PROGRAM Stn052_20_ReceivingBreakStopsGrn
VAR
	
//(1 omitted intentially, 3LnSw using this location)	
//		.fbBreakStop[1].iBufferFull :=  <0,1,0>TIIB[N21S00 (AL1332)]^N21S03 (AL2341)^TxPDO^input byte 2;
//		.fbBreakStop[1].iPuckPresent :=  <0,1,0>TIIB[N21S00 (AL1332)]^N21S03 (AL2341)^TxPDO^input byte 0;
//		.fbBreakStop[1].oStopLower :=  <0,1,4>TIIB[N21S00 (AL1332)]^N21S02 (EX260)^RxPDO^output byte 0;
//(3 omitted because the output byte overlaps 2 PLC projects, these are linked in Stn053)
//		.fbBreakStop[31].oStopLower :=  <0,1,0>TIIB[N32S00 (AL1332)]^N32S02 (EX260)^RxPDO^output byte 0;
//		.fbBreakStop[32].oStopLower :=  <0,1,1>TIIB[N32S00 (AL1332)]^N32S02 (EX260)^RxPDO^output byte 0;
//		.fbBreakStop[33].oStopLower :=  <0,1,2>TIIB[N32S00 (AL1332)]^N32S02 (EX260)^RxPDO^output byte 0'}	

	{attribute 'TcLinkToOSO' := '.fbBreakStop[2].iBufferFull :=  <0,1,1>TIIB[N21S00 (AL1332)]^N21S03 (AL2341)^TxPDO^input byte 2;
		.fbBreakStop[2].iPuckPresent :=  <0,1,1>TIIB[N21S00 (AL1332)]^N21S03 (AL2341)^TxPDO^input byte 0;
		.fbBreakStop[2].oStopLower :=  <0,1,5>TIIB[N21S00 (AL1332)]^N21S02 (EX260)^RxPDO^output byte 0;
		.fbBreakStop[3].iBufferFull :=  <0,1,0>TIIB[N21S00 (AL1332)]^N21S05 (AL2341)^TxPDO^input byte 2;
		.fbBreakStop[3].iPuckPresent :=  <0,1,0>TIIB[N21S00 (AL1332)]^N21S05 (AL2341)^TxPDO^input byte 0;
		.fbBreakStop[3].oStopLower :=  <0,1,6>TIIB[N21S00 (AL1332)]^N21S02 (EX260)^RxPDO^output byte 0;
		.fbBreakStop[4].iBufferFull :=  <0,1,0>TIIB[N26S00 (AL1332)]^N26S01 (AL2341)^TxPDO^input byte 2;
		.fbBreakStop[4].iPuckPresent :=  <0,1,0>TIIB[N26S00 (AL1332)]^N26S01 (AL2341)^TxPDO^input byte 0;
		.fbBreakStop[4].oStopLower :=  <0,1,0>TIIB[N26S00 (AL1332)]^N26S05 (EX260)^RxPDO^output byte 0;
		.fbBreakStop[5].iBufferFull :=  <0,1,2>TIIB[N26S00 (AL1332)]^N26S01 (AL2341)^TxPDO^input byte 2;
		.fbBreakStop[5].iPuckPresent :=  <0,1,2>TIIB[N26S00 (AL1332)]^N26S01 (AL2341)^TxPDO^input byte 0;
		.fbBreakStop[5].oStopLower :=  <0,1,1>TIIB[N26S00 (AL1332)]^N26S05 (EX260)^RxPDO^output byte 0;
		.fbBreakStop[6].iBufferFull :=  <0,1,3>TIIB[N26S00 (AL1332)]^N26S01 (AL2341)^TxPDO^input byte 2;
		.fbBreakStop[6].iPuckPresent :=  <0,1,3>TIIB[N26S00 (AL1332)]^N26S01 (AL2341)^TxPDO^input byte 0;
		.fbBreakStop[6].oStopLower :=  <0,1,4>TIIB[N26S00 (AL1332)]^N26S05 (EX260)^RxPDO^output byte 0;
		.fbBreakStop[7].iBufferFull :=  <0,1,4>TIIB[N26S00 (AL1332)]^N26S01 (AL2341)^TxPDO^input byte 2;
		.fbBreakStop[7].iPuckPresent :=  <0,1,4>TIIB[N26S00 (AL1332)]^N26S01 (AL2341)^TxPDO^input byte 0;
		.fbBreakStop[7].oStopLower :=  <0,1,5>TIIB[N26S00 (AL1332)]^N26S05 (EX260)^RxPDO^output byte 0;
		.fbBreakStop[8].iBufferFull :=  <0,1,0>TIIB[N26S00 (AL1332)]^N26S03 (AL2341)^TxPDO^input byte 2;
		.fbBreakStop[8].iPuckPresent :=  <0,1,0>TIIB[N26S00 (AL1332)]^N26S03 (AL2341)^TxPDO^input byte 0;
		.fbBreakStop[8].oStopLower :=  <0,1,0>TIIB[N26S00 (AL1332)]^N26S06 (EX260)^RxPDO^output byte 0;
		.fbBreakStop[9].iBufferFull :=  <0,1,2>TIIB[N26S00 (AL1332)]^N26S03 (AL2341)^TxPDO^input byte 2;
		.fbBreakStop[9].iPuckPresent :=  <0,1,2>TIIB[N26S00 (AL1332)]^N26S03 (AL2341)^TxPDO^input byte 0;
		.fbBreakStop[9].oStopLower :=  <0,1,1>TIIB[N26S00 (AL1332)]^N26S06 (EX260)^RxPDO^output byte 0;
		.fbBreakStop[10].iBufferFull :=  <0,1,3>TIIB[N26S00 (AL1332)]^N26S03 (AL2341)^TxPDO^input byte 2;
		.fbBreakStop[10].iPuckPresent :=  <0,1,3>TIIB[N26S00 (AL1332)]^N26S03 (AL2341)^TxPDO^input byte 0;
		.fbBreakStop[10].oStopLower :=  <0,1,4>TIIB[N26S00 (AL1332)]^N26S06 (EX260)^RxPDO^output byte 0;
		.fbBreakStop[11].iBufferFull :=  <0,1,4>TIIB[N26S00 (AL1332)]^N26S03 (AL2341)^TxPDO^input byte 2;
		.fbBreakStop[11].iPuckPresent :=  <0,1,4>TIIB[N26S00 (AL1332)]^N26S03 (AL2341)^TxPDO^input byte 0;
		.fbBreakStop[11].oStopLower :=  <0,1,5>TIIB[N26S00 (AL1332)]^N26S06 (EX260)^RxPDO^output byte 0;
		.fbBreakStop[12].iBufferFull :=  <0,1,0>TIIB[N27S00 (AL1332)]^N27S01 (AL2341)^TxPDO^input byte 2;
		.fbBreakStop[12].iPuckPresent :=  <0,1,0>TIIB[N27S00 (AL1332)]^N27S01 (AL2341)^TxPDO^input byte 0;
		.fbBreakStop[12].oStopLower :=  <0,1,0>TIIB[N27S00 (AL1332)]^N27S05 (EX260)^RxPDO^output byte 0;
		.fbBreakStop[13].iBufferFull :=  <0,1,2>TIIB[N27S00 (AL1332)]^N27S01 (AL2341)^TxPDO^input byte 2;
		.fbBreakStop[13].iPuckPresent :=  <0,1,2>TIIB[N27S00 (AL1332)]^N27S01 (AL2341)^TxPDO^input byte 0;
		.fbBreakStop[13].oStopLower :=  <0,1,1>TIIB[N27S00 (AL1332)]^N27S05 (EX260)^RxPDO^output byte 0;
		.fbBreakStop[14].iBufferFull :=  <0,1,3>TIIB[N27S00 (AL1332)]^N27S01 (AL2341)^TxPDO^input byte 2;
		.fbBreakStop[14].iPuckPresent :=  <0,1,3>TIIB[N27S00 (AL1332)]^N27S01 (AL2341)^TxPDO^input byte 0;
		.fbBreakStop[14].oStopLower :=  <0,1,4>TIIB[N27S00 (AL1332)]^N27S05 (EX260)^RxPDO^output byte 0;
		.fbBreakStop[15].iBufferFull :=  <0,1,4>TIIB[N27S00 (AL1332)]^N27S01 (AL2341)^TxPDO^input byte 2;
		.fbBreakStop[15].iPuckPresent :=  <0,1,4>TIIB[N27S00 (AL1332)]^N27S01 (AL2341)^TxPDO^input byte 0;
		.fbBreakStop[15].oStopLower :=  <0,1,5>TIIB[N27S00 (AL1332)]^N27S05 (EX260)^RxPDO^output byte 0;
		.fbBreakStop[16].iBufferFull :=  <0,1,0>TIIB[N27S00 (AL1332)]^N27S03 (AL2341)^TxPDO^input byte 2;
		.fbBreakStop[16].iPuckPresent :=  <0,1,0>TIIB[N27S00 (AL1332)]^N27S03 (AL2341)^TxPDO^input byte 0;
		.fbBreakStop[16].oStopLower :=  <0,1,0>TIIB[N27S00 (AL1332)]^N27S06 (EX260)^RxPDO^output byte 0;
		.fbBreakStop[17].iBufferFull :=  <0,1,2>TIIB[N27S00 (AL1332)]^N27S03 (AL2341)^TxPDO^input byte 2;
		.fbBreakStop[17].iPuckPresent :=  <0,1,2>TIIB[N27S00 (AL1332)]^N27S03 (AL2341)^TxPDO^input byte 0;
		.fbBreakStop[17].oStopLower :=  <0,1,1>TIIB[N27S00 (AL1332)]^N27S06 (EX260)^RxPDO^output byte 0;
		.fbBreakStop[18].iBufferFull :=  <0,1,3>TIIB[N27S00 (AL1332)]^N27S03 (AL2341)^TxPDO^input byte 2;
		.fbBreakStop[18].iPuckPresent :=  <0,1,3>TIIB[N27S00 (AL1332)]^N27S03 (AL2341)^TxPDO^input byte 0;
		.fbBreakStop[18].oStopLower :=  <0,1,4>TIIB[N27S00 (AL1332)]^N27S06 (EX260)^RxPDO^output byte 0;
		.fbBreakStop[19].iBufferFull :=  <0,1,4>TIIB[N27S00 (AL1332)]^N27S03 (AL2341)^TxPDO^input byte 0;
		.fbBreakStop[19].iPuckPresent :=  <0,1,4>TIIB[N27S00 (AL1332)]^N27S03 (AL2341)^TxPDO^input byte 2;
		.fbBreakStop[19].oStopLower :=  <0,1,5>TIIB[N27S00 (AL1332)]^N27S06 (EX260)^RxPDO^output byte 0;
		.fbBreakStop[20].iBufferFull :=  <0,1,3>TIIB[N28S00 (AL1332)]^N28S01 (AL2341)^TxPDO^input byte 2;
		.fbBreakStop[20].iPuckPresent :=  <0,1,3>TIIB[N28S00 (AL1332)]^N28S01 (AL2341)^TxPDO^input byte 0;
		.fbBreakStop[20].oStopLower :=  <0,1,4>TIIB[N28S00 (AL1332)]^N28S05 (EX260)^RxPDO^output byte 0;
		.fbBreakStop[21].iBufferFull :=  <0,1,4>TIIB[N28S00 (AL1332)]^N28S01 (AL2341)^TxPDO^input byte 2;
		.fbBreakStop[21].iPuckPresent :=  <0,1,4>TIIB[N28S00 (AL1332)]^N28S01 (AL2341)^TxPDO^input byte 0;
		.fbBreakStop[21].oStopLower :=  <0,1,5>TIIB[N28S00 (AL1332)]^N28S05 (EX260)^RxPDO^output byte 0;
		.fbBreakStop[22].iBufferFull :=  <0,1,3>TIIB[N28S00 (AL1332)]^N28S03 (AL2341)^TxPDO^input byte 2;
		.fbBreakStop[22].iPuckPresent :=  <0,1,3>TIIB[N28S00 (AL1332)]^N28S03 (AL2341)^TxPDO^input byte 0;
		.fbBreakStop[22].oStopLower :=  <0,1,4>TIIB[N28S00 (AL1332)]^N28S06 (EX260)^RxPDO^output byte 0;
		.fbBreakStop[23].iBufferFull :=  <0,1,4>TIIB[N28S00 (AL1332)]^N28S03 (AL2341)^TxPDO^input byte 2;
		.fbBreakStop[23].iPuckPresent :=  <0,1,4>TIIB[N28S00 (AL1332)]^N28S03 (AL2341)^TxPDO^input byte 0;
		.fbBreakStop[23].oStopLower :=  <0,1,5>TIIB[N28S00 (AL1332)]^N28S06 (EX260)^RxPDO^output byte 0;
		.fbBreakStop[24].iBufferFull :=  <0,1,0>TIIB[N31S00 (AL1332)]^N31S01 (AL2341)^TxPDO^input byte 2;
		.fbBreakStop[24].iPuckPresent :=  <0,1,0>TIIB[N31S00 (AL1332)]^N31S01 (AL2341)^TxPDO^input byte 0;
		.fbBreakStop[24].oStopLower :=  <0,1,0>TIIB[N31S00 (AL1332)]^N31S02 (EX260)^RxPDO^output byte 0;
		.fbBreakStop[25].iBufferFull :=  <0,1,1>TIIB[N31S00 (AL1332)]^N31S01 (AL2341)^TxPDO^input byte 2;
		.fbBreakStop[25].iPuckPresent :=  <0,1,1>TIIB[N31S00 (AL1332)]^N31S01 (AL2341)^TxPDO^input byte 0;
		.fbBreakStop[25].oStopLower :=  <0,1,1>TIIB[N31S00 (AL1332)]^N31S02 (EX260)^RxPDO^output byte 0;
		.fbBreakStop[26].iBufferFull :=  <0,1,2>TIIB[N31S00 (AL1332)]^N31S01 (AL2341)^TxPDO^input byte 2;
		.fbBreakStop[26].iPuckPresent :=  <0,1,2>TIIB[N31S00 (AL1332)]^N31S01 (AL2341)^TxPDO^input byte 0;
		.fbBreakStop[26].oStopLower :=  <0,1,2>TIIB[N31S00 (AL1332)]^N31S02 (EX260)^RxPDO^output byte 0;
		.fbBreakStop[27].iBufferFull :=  <0,1,0>TIIB[N31S00 (AL1332)]^N31S03 (AL2341)^TxPDO^input byte 2;
		.fbBreakStop[27].iPuckPresent :=  <0,1,0>TIIB[N31S00 (AL1332)]^N31S03 (AL2341)^TxPDO^input byte 0;
		.fbBreakStop[27].oStopLower :=  <0,1,3>TIIB[N31S00 (AL1332)]^N31S02 (EX260)^RxPDO^output byte 0;
		.fbBreakStop[28].iBufferFull :=  <0,1,1>TIIB[N31S00 (AL1332)]^N31S03 (AL2341)^TxPDO^input byte 2;
		.fbBreakStop[28].iPuckPresent :=  <0,1,1>TIIB[N31S00 (AL1332)]^N31S03 (AL2341)^TxPDO^input byte 0;
		.fbBreakStop[28].oStopLower :=  <0,1,4>TIIB[N31S00 (AL1332)]^N31S02 (EX260)^RxPDO^output byte 0;
		.fbBreakStop[29].iBufferFull :=  <0,1,2>TIIB[N31S00 (AL1332)]^N31S03 (AL2341)^TxPDO^input byte 2;
		.fbBreakStop[29].iPuckPresent :=  <0,1,2>TIIB[N31S00 (AL1332)]^N31S03 (AL2341)^TxPDO^input byte 0;
		.fbBreakStop[29].oStopLower :=  <0,1,5>TIIB[N31S00 (AL1332)]^N31S02 (EX260)^RxPDO^output byte 0;
		.fbBreakStop[30].iBufferFull :=  <0,1,0>TIIB[N31S00 (AL1332)]^N31S05 (AL2341)^TxPDO^input byte 2;
		.fbBreakStop[30].iPuckPresent :=  <0,1,0>TIIB[N31S00 (AL1332)]^N31S05 (AL2341)^TxPDO^input byte 0;
		.fbBreakStop[30].oStopLower :=  <0,1,6>TIIB[N31S00 (AL1332)]^N31S02 (EX260)^RxPDO^output byte 0;
		.fbBreakStop[31].iBufferFull :=  <0,1,0>TIIB[N31S00 (AL1332)]^N31S07 (AL2341)^TxPDO^input byte 2;
		.fbBreakStop[31].iPuckPresent :=  <0,1,0>TIIB[N31S00 (AL1332)]^N31S07 (AL2341)^TxPDO^input byte 0;
		.fbBreakStop[32].iBufferFull :=  <0,1,1>TIIB[N31S00 (AL1332)]^N31S07 (AL2341)^TxPDO^input byte 2;
		.fbBreakStop[32].iPuckPresent :=  <0,1,1>TIIB[N31S00 (AL1332)]^N31S07 (AL2341)^TxPDO^input byte 0;
		.fbBreakStop[33].iBufferFull :=  <0,1,0>TIIB[N32S00 (AL1332)]^N32S01 (AL2341)^TxPDO^input byte 2;
		.fbBreakStop[33].iPuckPresent :=  <0,1,0>TIIB[N32S00 (AL1332)]^N32S01 (AL2341)^TxPDO^input byte 0'}
	fbBreakStopGroup: FB_BreakStopGroup;
	
	i: DINT;
	
END_VAR

//  This code instantiates a component that is implimented as a common function block
//    Note that I/O is linked directly to I/O variables inside the named instance

//  combine running state of any multiple conveyors in a break stop here.
// motor control status here - Green conv  

gStn052_20_ReceivingBreakStopsGrn.ConvRunning[02] := gConsumed_SafetyInterfaceConv.MtrRunning.Enc054Mtr01;
gStn052_20_ReceivingBreakStopsGrn.ConvRunning[03] := gConsumed_SafetyInterfaceConv.MtrRunning.Enc054Mtr01;
gStn052_20_ReceivingBreakStopsGrn.ConvRunning[04] := gConsumed_SafetyInterfaceConv.MtrRunning.Enc054Mtr01;
gStn052_20_ReceivingBreakStopsGrn.ConvRunning[05] := gConsumed_SafetyInterfaceConv.MtrRunning.Enc054Mtr01;
gStn052_20_ReceivingBreakStopsGrn.ConvRunning[06] := gConsumed_SafetyInterfaceConv.MtrRunning.Enc054Mtr01;
gStn052_20_ReceivingBreakStopsGrn.ConvRunning[07] := gConsumed_SafetyInterfaceConv.MtrRunning.Enc054Mtr01;
gStn052_20_ReceivingBreakStopsGrn.ConvRunning[08] := gConsumed_SafetyInterfaceConv.MtrRunning.Enc054Mtr01;
gStn052_20_ReceivingBreakStopsGrn.ConvRunning[09] := gConsumed_SafetyInterfaceConv.MtrRunning.Enc054Mtr01 AND gConsumed_SafetyInterfaceConv.MtrRunning.Enc054Mtr02;
gStn052_20_ReceivingBreakStopsGrn.ConvRunning[10] := gConsumed_SafetyInterfaceConv.MtrRunning.Enc054Mtr02;
gStn052_20_ReceivingBreakStopsGrn.ConvRunning[11] := gConsumed_SafetyInterfaceConv.MtrRunning.Enc054Mtr02;
gStn052_20_ReceivingBreakStopsGrn.ConvRunning[12] := gConsumed_SafetyInterfaceConv.MtrRunning.Enc054Mtr02;
gStn052_20_ReceivingBreakStopsGrn.ConvRunning[13] := gConsumed_SafetyInterfaceConv.MtrRunning.Enc054Mtr02;
gStn052_20_ReceivingBreakStopsGrn.ConvRunning[14] := gConsumed_SafetyInterfaceConv.MtrRunning.Enc054Mtr02;
gStn052_20_ReceivingBreakStopsGrn.ConvRunning[15] := gConsumed_SafetyInterfaceConv.MtrRunning.Enc054Mtr02;
gStn052_20_ReceivingBreakStopsGrn.ConvRunning[16] := gConsumed_SafetyInterfaceConv.MtrRunning.Enc054Mtr02;
gStn052_20_ReceivingBreakStopsGrn.ConvRunning[17] := gConsumed_SafetyInterfaceConv.MtrRunning.Enc054Mtr02 AND gConsumed_SafetyInterfaceConv.MtrRunning.Enc054Mtr03;
gStn052_20_ReceivingBreakStopsGrn.ConvRunning[18] := gConsumed_SafetyInterfaceConv.MtrRunning.Enc054Mtr03;
gStn052_20_ReceivingBreakStopsGrn.ConvRunning[19] := gConsumed_SafetyInterfaceConv.MtrRunning.Enc054Mtr03;
gStn052_20_ReceivingBreakStopsGrn.ConvRunning[20] := gConsumed_SafetyInterfaceConv.MtrRunning.Enc054Mtr03;
gStn052_20_ReceivingBreakStopsGrn.ConvRunning[21] := gConsumed_SafetyInterfaceConv.MtrRunning.Enc054Mtr03;
gStn052_20_ReceivingBreakStopsGrn.ConvRunning[22] := gConsumed_SafetyInterfaceConv.MtrRunning.Enc054Mtr03;
gStn052_20_ReceivingBreakStopsGrn.ConvRunning[23] := gConsumed_SafetyInterfaceConv.MtrRunning.Enc054Mtr03 AND gConsumed_SafetyInterfaceConv.MtrRunning.Enc055Mtr01;
gStn052_20_ReceivingBreakStopsGrn.ConvRunning[24] := gConsumed_SafetyInterfaceConv.MtrRunning.Enc055Mtr01;
gStn052_20_ReceivingBreakStopsGrn.ConvRunning[25] := gConsumed_SafetyInterfaceConv.MtrRunning.Enc055Mtr01;
gStn052_20_ReceivingBreakStopsGrn.ConvRunning[26] := gConsumed_SafetyInterfaceConv.MtrRunning.Enc055Mtr01;
gStn052_20_ReceivingBreakStopsGrn.ConvRunning[27] := gConsumed_SafetyInterfaceConv.MtrRunning.Enc055Mtr01;
gStn052_20_ReceivingBreakStopsGrn.ConvRunning[28] := gConsumed_SafetyInterfaceConv.MtrRunning.Enc055Mtr01;
gStn052_20_ReceivingBreakStopsGrn.ConvRunning[29] := gConsumed_SafetyInterfaceConv.MtrRunning.Enc055Mtr01 AND gConsumed_SafetyInterfaceConv.MtrRunning.Enc055Mtr02;;
gStn052_20_ReceivingBreakStopsGrn.ConvRunning[30] := gConsumed_SafetyInterfaceConv.MtrRunning.Enc055Mtr02;
gStn052_20_ReceivingBreakStopsGrn.ConvRunning[31] := gConsumed_SafetyInterfaceConv.MtrRunning.Enc055Mtr02;
gStn052_20_ReceivingBreakStopsGrn.ConvRunning[32] := gConsumed_SafetyInterfaceConv.MtrRunning.Enc055Mtr02;
gStn052_20_ReceivingBreakStopsGrn.ConvRunning[33] := gConsumed_SafetyInterfaceConv.MtrRunning.Enc055Mtr02 AND gConsumed_SafetyInterfaceConv.Stn053PLCData[0].10;


fbBreakStopGroup(
	pStn := ADR(gStn052),
	pCmp := ADR(gStn052_20_ReceivingBreakStopsGrn),
	pStateTraceBuffer := ADR(gStn052_StateTraceBuffer),
	pStateTraceFifo := ADR(gStn052_StateTraceFifo),
	pStats := ADR(gStn052_02_Stats),
);

//Producing lower stop request to station 053 for shared valve bank
gProduced_Stn052ToSafetyInterface.Stn052PLCData[0].0 := gStn052_20_ReceivingBreakStopsGrn.LowerStopReq[31];
gProduced_Stn052ToSafetyInterface.Stn052PLCData[0].1 := gStn052_20_ReceivingBreakStopsGrn.LowerStopReq[32];
gProduced_Stn052ToSafetyInterface.Stn052PLCData[0].2 := gStn052_20_ReceivingBreakStopsGrn.LowerStopReq[33];

END_PROGRAM

(* stored: Version 1.1.0.1, ProductVersion 3.1.4024.6
   POU Stn052_20_ReceivingBreakStopsGrn: Id {d8484e1c-93b3-4313-ba24-5299c1568373}, SpecialFunc None *)
